INTERFACE I_ParameterVisitor

METHOD VisitParameter
VAR_INPUT
	VisitingProperty : I_Parameter;
END_VAR
END_METHOD

END_INTERFACE

(* stored: Version 1.1.0.1, ProductVersion 3.1.4024.12
   Itf I_ParameterVisitor: Id {2b8d46db-1503-4c93-9b55-80e7a901db90}
   Method VisitParameter: Id {0ba9be72-c689-4093-bb8b-26759a8e218d} *)
